% RSLogix 500 project Sesion11_Tarea1_Josue Santana Robledo Corona.RSS, saved by version 8.40.00.08 %
PROJECT "UNTITLED"    % processor: MicroLogix 1200 %

PROGRAM FILES
  LAD 2 "MAIN"  6 rungs
  LAD 3 "ENTRADAS"  6 rungs
  LAD 4 "SALIDAS"  4 rungs
  LAD 5 "AUTOMATICO"  13 rungs
  LAD 6 "MANUAL"  4 rungs
  LAD 7 "HMI"  1 rungs
  LAD 8 "ALARMAS"  1 rungs
  LAD 9 "PARPADEOS"  5 rungs
  LAD 10 "LS"  2 rungs

DATA FILES
  O0 OUTPUT  4 elements
  I1 INPUT  4 elements
  S2 STATUS  66 elements
  B3 BINARY  3 elements
  T4 TIMER  5 elements
  C5 COUNTER  2 elements
  R6 CONTROL  1 elements
  N7 INTEGER  1 elements
  F8 FLOAT  1 elements

LADDER 2 "MAIN"
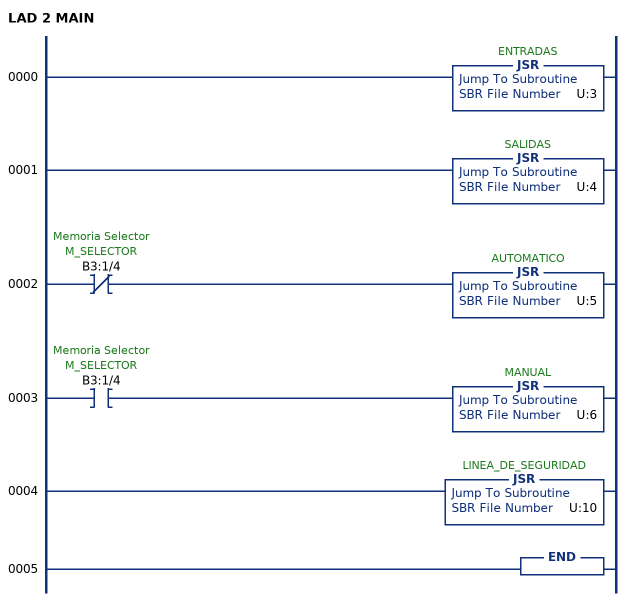
% Rung: 0 %
SOR JSR U:3 EOR
%   U:3  ENTRADAS %
% Rung: 1 %
SOR JSR U:4 EOR
%   U:4  SALIDAS %
% Rung: 2 %
SOR XIO B3:1/4 JSR U:5 EOR
%   B3:1/4  M_SELECTOR  "Memoria Selector" %
%   U:5  AUTOMATICO %
% Rung: 3 %
SOR XIC B3:1/4 JSR U:6 EOR
%   B3:1/4  M_SELECTOR  "Memoria Selector" %
%   U:6  MANUAL %
% Rung: 4 %
SOR JSR U:10 EOR
%   U:10  LINEA_DE_SEGURIDAD %
% Rung: 5 %
SOR END EOR

LADDER 3 "ENTRADAS"
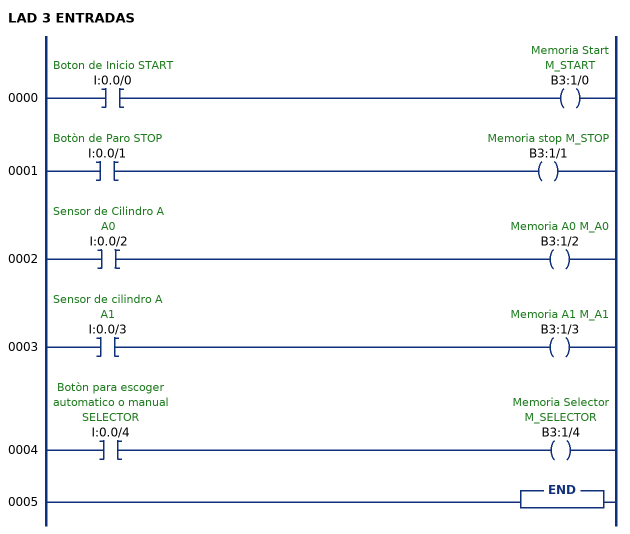
% Rung: 0 %
SOR XIC I:0.0/0 OTE B3:1/0 EOR
%   I:0.0/0  START  "Boton de Inicio" %
%   B3:1/0  M_START  "Memoria Start" %
% Rung: 1 %
SOR XIC I:0.0/1 OTE B3:1/1 EOR
%   I:0.0/1  STOP  "Botòn de Paro" %
%   B3:1/1  M_STOP  "Memoria stop" %
% Rung: 2 %
SOR XIC I:0.0/2 OTE B3:1/2 EOR
%   I:0.0/2  A0  "Sensor de Cilindro A" %
%   B3:1/2  M_A0  "Memoria A0" %
% Rung: 3 %
SOR XIC I:0.0/3 OTE B3:1/3 EOR
%   I:0.0/3  A1  "Sensor de cilindro A" %
%   B3:1/3  M_A1  "Memoria A1" %
% Rung: 4 %
SOR XIC I:0.0/4 OTE B3:1/4 EOR
%   I:0.0/4  SELECTOR  "Botòn para escoger automatico o manual" %
%   B3:1/4  M_SELECTOR  "Memoria Selector" %
% Rung: 5 %
SOR END EOR

LADDER 4 "SALIDAS"
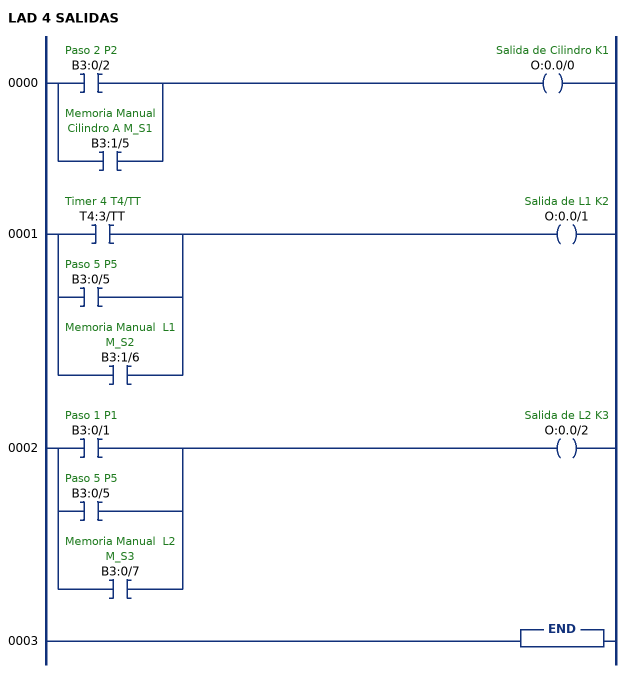
% Rung: 0 %
SOR BST XIC B3:0/2 NXB XIC B3:1/5 BND OTE O:0.0/0 EOR
%   B3:0/2  P2  "Paso 2" %
%   B3:1/5  M_S1  "Memoria Manual Cilindro A" %
%   O:0.0/0  K1  "Salida de Cilindro" %
% Rung: 1 %
SOR BST XIC T4:3/TT NXB XIC B3:0/5 NXB XIC B3:1/6 BND OTE O:0.0/1 EOR
%   T4:3  T4  "Timer 4" %
%   B3:0/5  P5  "Paso 5" %
%   B3:1/6  M_S2  "Memoria Manual  L1" %
%   O:0.0/1  K2  "Salida de L1" %
% Rung: 2 %
SOR BST XIC B3:0/1 NXB XIC B3:0/5 NXB XIC B3:0/7 BND OTE O:0.0/2 EOR
%   B3:0/1  P1  "Paso 1" %
%   B3:0/5  P5  "Paso 5" %
%   B3:0/7  M_S3  "Memoria Manual  L2" %
%   O:0.0/2  K3  "Salida de L2" %
% Rung: 3 %
SOR END EOR

LADDER 5 "AUTOMATICO"
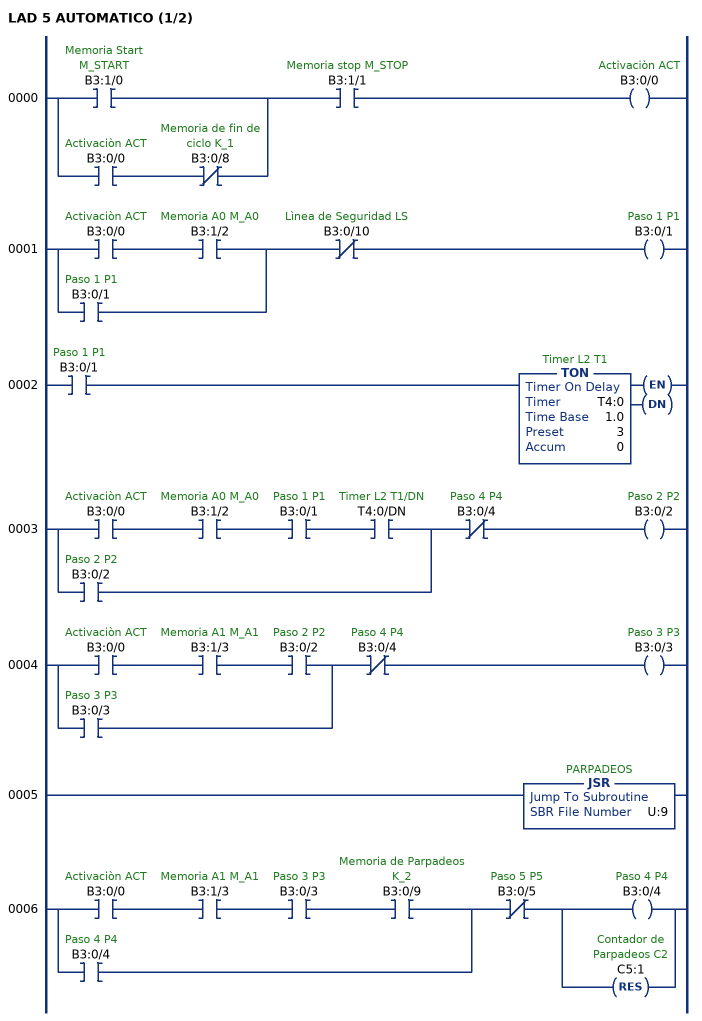
% Rung: 0 %
SOR BST XIC B3:1/0 NXB XIC B3:0/0 XIO B3:0/8 BND XIC B3:1/1 OTE B3:0/0 EOR
%   B3:1/0  M_START  "Memoria Start" %
%   B3:0/0  ACT  "Activaciòn" %
%   B3:0/8  K_1  "Memoria de fin de ciclo" %
%   B3:1/1  M_STOP  "Memoria stop" %
% Rung: 1 %
SOR BST XIC B3:0/0 XIC B3:1/2 NXB XIC B3:0/1 BND XIO B3:0/10 OTE B3:0/1 EOR
%   B3:0/0  ACT  "Activaciòn" %
%   B3:1/2  M_A0  "Memoria A0" %
%   B3:0/1  P1  "Paso 1" %
%   B3:0/10  LS  "Lìnea de Seguridad" %
% Rung: 2 %
SOR XIC B3:0/1 TON T4:0 1.0 3 0 EOR
%   B3:0/1  P1  "Paso 1" %
%   T4:0  T1  "Timer L2" %
% Rung: 3 %
SOR BST XIC B3:0/0 XIC B3:1/2 XIC B3:0/1 XIC T4:0/DN NXB XIC B3:0/2 BND XIO B3:0/4 OTE B3:0/2 EOR
%   B3:0/0  ACT  "Activaciòn" %
%   B3:1/2  M_A0  "Memoria A0" %
%   B3:0/1  P1  "Paso 1" %
%   T4:0  T1  "Timer L2" %
%   B3:0/2  P2  "Paso 2" %
%   B3:0/4  P4  "Paso 4" %
% Rung: 4 %
SOR BST XIC B3:0/0 XIC B3:1/3 XIC B3:0/2 NXB XIC B3:0/3 BND XIO B3:0/4 OTE B3:0/3 EOR
%   B3:0/0  ACT  "Activaciòn" %
%   B3:1/3  M_A1  "Memoria A1" %
%   B3:0/2  P2  "Paso 2" %
%   B3:0/3  P3  "Paso 3" %
%   B3:0/4  P4  "Paso 4" %
% Rung: 5 %
SOR JSR U:9 EOR
%   U:9  PARPADEOS %
% Rung: 6 %
SOR BST XIC B3:0/0 XIC B3:1/3 XIC B3:0/3 XIC B3:0/9 NXB XIC B3:0/4 BND XIO B3:0/5 BST OTE B3:0/4 NXB RES C5:1 BND EOR
%   B3:0/0  ACT  "Activaciòn" %
%   B3:1/3  M_A1  "Memoria A1" %
%   B3:0/3  P3  "Paso 3" %
%   B3:0/9  K_2  "Memoria de Parpadeos" %
%   B3:0/4  P4  "Paso 4" %
%   B3:0/5  P5  "Paso 5" %
%   C5:1  C2  "Contador de Parpadeos" %

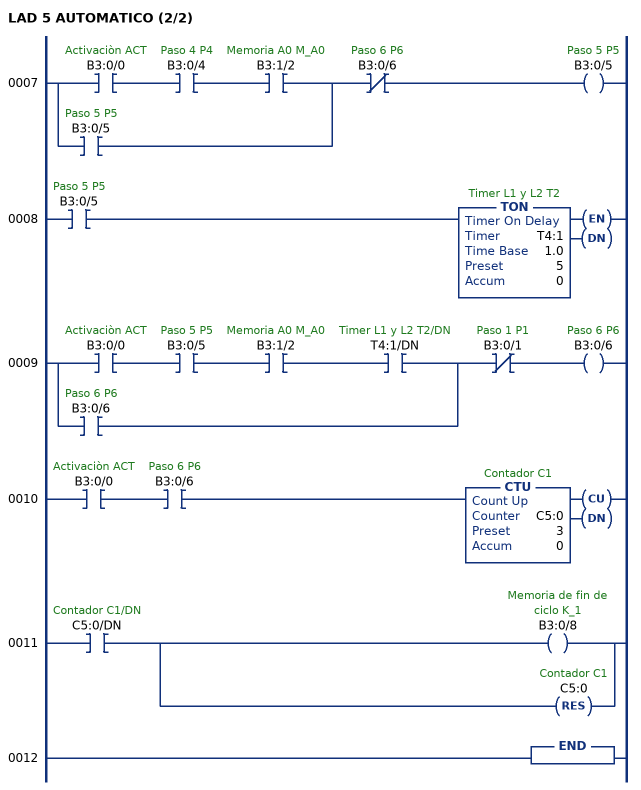
% Rung: 7 %
SOR BST XIC B3:0/0 XIC B3:0/4 XIC B3:1/2 NXB XIC B3:0/5 BND XIO B3:0/6 OTE B3:0/5 EOR
%   B3:0/0  ACT  "Activaciòn" %
%   B3:0/4  P4  "Paso 4" %
%   B3:1/2  M_A0  "Memoria A0" %
%   B3:0/5  P5  "Paso 5" %
%   B3:0/6  P6  "Paso 6" %
% Rung: 8 %
SOR XIC B3:0/5 TON T4:1 1.0 5 0 EOR
%   B3:0/5  P5  "Paso 5" %
%   T4:1  T2  "Timer L1 y L2" %
% Rung: 9 %
SOR BST XIC B3:0/0 XIC B3:0/5 XIC B3:1/2 XIC T4:1/DN NXB XIC B3:0/6 BND XIO B3:0/1 OTE B3:0/6 EOR
%   B3:0/0  ACT  "Activaciòn" %
%   B3:0/5  P5  "Paso 5" %
%   B3:1/2  M_A0  "Memoria A0" %
%   T4:1  T2  "Timer L1 y L2" %
%   B3:0/6  P6  "Paso 6" %
%   B3:0/1  P1  "Paso 1" %
% Rung: 10 %
SOR XIC B3:0/0 XIC B3:0/6 CTU C5:0 3 0 EOR
%   B3:0/0  ACT  "Activaciòn" %
%   B3:0/6  P6  "Paso 6" %
%   C5:0  C1  "Contador" %
% Rung: 11 %
SOR XIC C5:0/DN BST OTE B3:0/8 NXB RES C5:0 BND EOR
%   C5:0  C1  "Contador" %
%   B3:0/8  K_1  "Memoria de fin de ciclo" %
% Rung: 12 %
SOR END EOR

LADDER 6 "MANUAL"
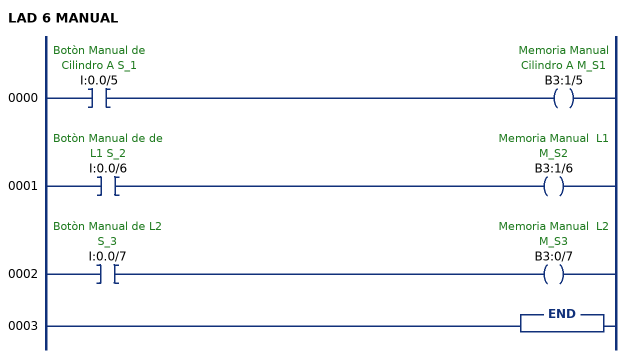
% Rung: 0 %
SOR XIC I:0.0/5 OTE B3:1/5 EOR
%   I:0.0/5  S_1  "Botòn Manual de Cilindro A" %
%   B3:1/5  M_S1  "Memoria Manual Cilindro A" %
% Rung: 1 %
SOR XIC I:0.0/6 OTE B3:1/6 EOR
%   I:0.0/6  S_2  "Botòn Manual de de L1" %
%   B3:1/6  M_S2  "Memoria Manual  L1" %
% Rung: 2 %
SOR XIC I:0.0/7 OTE B3:0/7 EOR
%   I:0.0/7  S_3  "Botòn Manual de L2" %
%   B3:0/7  M_S3  "Memoria Manual  L2" %
% Rung: 3 %
SOR END EOR

LADDER 9 "PARPADEOS"
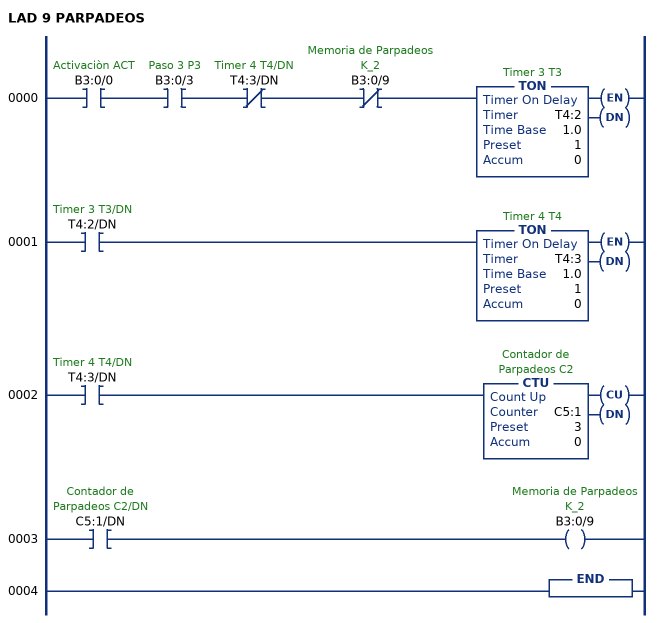
% Rung: 0 %
SOR XIC B3:0/0 XIC B3:0/3 XIO T4:3/DN XIO B3:0/9 TON T4:2 1.0 1 0 EOR
%   B3:0/0  ACT  "Activaciòn" %
%   B3:0/3  P3  "Paso 3" %
%   T4:3  T4  "Timer 4" %
%   B3:0/9  K_2  "Memoria de Parpadeos" %
%   T4:2  T3  "Timer 3" %
% Rung: 1 %
SOR XIC T4:2/DN TON T4:3 1.0 1 0 EOR
%   T4:2  T3  "Timer 3" %
%   T4:3  T4  "Timer 4" %
% Rung: 2 %
SOR XIC T4:3/DN CTU C5:1 3 0 EOR
%   T4:3  T4  "Timer 4" %
%   C5:1  C2  "Contador de Parpadeos" %
% Rung: 3 %
SOR XIC C5:1/DN OTE B3:0/9 EOR
%   C5:1  C2  "Contador de Parpadeos" %
%   B3:0/9  K_2  "Memoria de Parpadeos" %
% Rung: 4 %
SOR END EOR

LADDER 10 "LS"
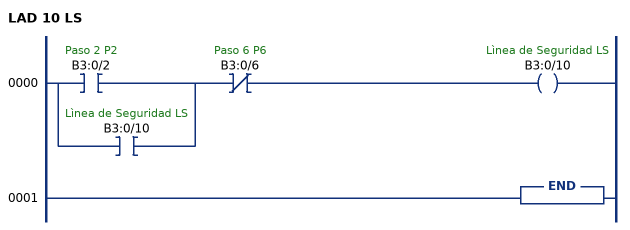
% Rung: 0 %
SOR BST XIC B3:0/2 NXB XIC B3:0/10 BND XIO B3:0/6 OTE B3:0/10 EOR
%   B3:0/2  P2  "Paso 2" %
%   B3:0/10  LS  "Lìnea de Seguridad" %
%   B3:0/6  P6  "Paso 6" %
% Rung: 1 %
SOR END EOR

DATA TABLE (non-zero values as saved)
DATA B3
% B3:0 % 0X0200 0X0000 0X0000
DATA T4
% .PRE .ACC %
% T4:0 % 3 0
% T4:1 % 5 0
% T4:2 % 1 0
% T4:3 % 1 0
DATA C5
% .PRE .ACC %
% C5:0 % 3 0
% C5:1 % 3 0
